TYPE ST_SubsystemBaseEmulation :
(**************************************************************************************
 * 	Application		:	BoxControl Framework
 *	Revision		:	$Revision: 404529 $
 *	Revision date	:	$Date: 2018-04-23 08:21:38 +0200 (Mo., 23 Apr 2018) $
 *	Last changed by	:	$Author: b7bolm $
 *	URL				:	$URL: http://almscdc.swisslog.com/repo/SWPD/Development/BoxControlFramework/20_Release/trunk/01_Software/BCF/BCF/JumpStart/20_Product/11_Emu/15_Subsystem/10_Lib/10_Conv/01_DUTs/ST_SubsystemBaseEmulation.TcDUT $
 *
 *	Purpose			:	Function interface - Contains data which is provided by the
 *						function or is input from other objects.
 *
 * ------------------------------------------------------------------------------------
 *	Copyright Swisslog [IP AG], Switzerland. All rights reserved.
 * 
 * ------------------------------------------------------------------------------------
 *	
 * 	Revision History: 
 *
 * 	VERSION			DATE			INITIALS			DESCRIPTION
 *	0.1				01.01.2001		swl					Example
 *
 **************************************************************************************)
STRUCT
	eITC_MsgType			: E_ITC_MsgTypeConv; // Last ITC message	
	rSubsystemDataReal		: REFERENCE TO ST_SubsystemData;
	SubsystemDataEmpty		: ST_SubsystemData;
	rSubsystemInterfaceReal	: REFERENCE TO ST_SubsystemInterface;
	SubsystemInterfaceEmpty : ST_SubsystemInterface;
	rSettingsSubsystemReal	: REFERENCE TO ST_CFG_Subsystem; // Element settings 	
	SettingsSubsystemEmpty  : ST_CFG_Subsystem;
	ERQ						: ST_ITC_ERQ;	
END_STRUCT
END_TYPE

(* stored: Version 1.1.0.1, ProductVersion 3.1.4022.12
   DUT ST_SubsystemBaseEmulation: Id {b8b1bc25-5279-4cc7-b370-18afddf5f234} *)
